ABB RobotStudio station: sesion1.rsstn

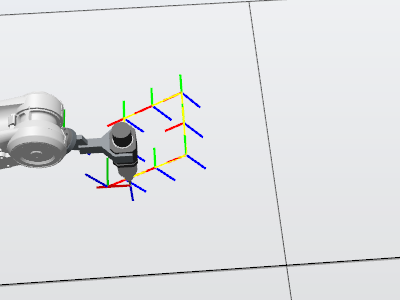
Station sesion1 (saved by RobotStudio 24.1.10713.1)
Controller Controlador1
  mechanical unit ROB_1: IRB140_6_81_C_03, 6 joints, base frame (0, 0, 0) mm
Layout (positions relative to the parent item):
  - IRB140_6_81_C_03 [mechanism, from %ABB.RobotStudio.Models.IRB140%\IRB140_6_81_C_G_03.rslib] at (0, 0, 0) mm; joint values [0, 0.0003, -0.1849, 0, 1.0922, 0] (rad or m)
  - MyTool [mechanism, from Training Objects\myTool.rslib] at (483.67, 0, 730.53) mm, rotated rx 180 ry 38 rz 180 deg
Attachment: MyTool is attached to IRB140_6_81_C_03 / Link6
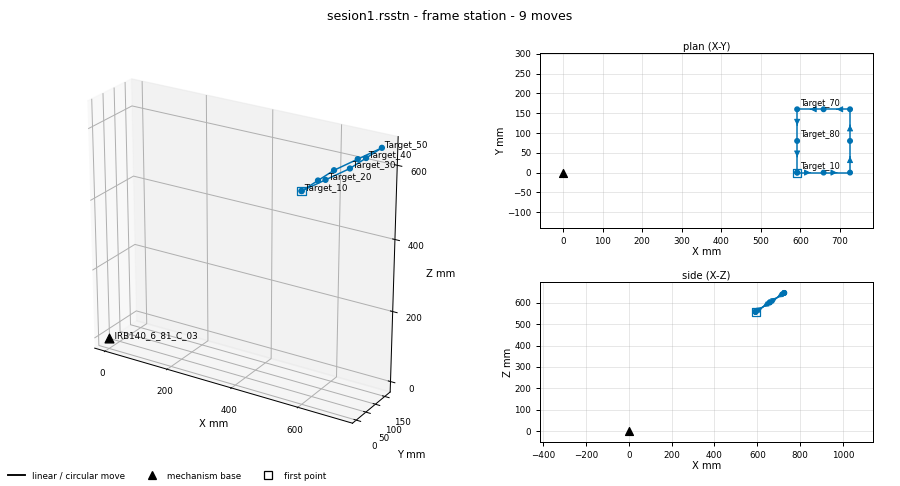
[picture p0: tool path of sesion1.rsstn in frame station, 9 of 9 moves have a stored position in this frame; points joined in program order, loops and branches not executed]
Targets, tools, work objects and paths stored in the station, written as RAPID:
! task T_ROB1
MODULE CalibData
  PERS tooldata MyTool:=[TRUE,[[31.792631019,0,229.638935148],[0.945518576,0,0.325568154,0]],[1,[0,0,1],[1,0,0,0],0,0,0]];
  TASK PERS wobjdata Workobject_1:=[FALSE,TRUE,"",[[550,0,530],[0.957921558,0,-0.287030119,0]],[[0,0,0],[1,0,0,0]]];
ENDMODULE

! task T_ROB1
MODULE Module1
  CONST robtarget Target_10:=[[50,0,0],[0,0,1,0],[0,-1,0,0],[9E+09,9E+09,9E+09,9E+09,9E+09,9E+09]];
  CONST robtarget Target_20:=[[130,0,0],[0,0,1,0],[0,0,-1,0],[9E+09,9E+09,9E+09,9E+09,9E+09,9E+09]];
  CONST robtarget Target_30:=[[210,0,0],[0,0,1,0],[-1,0,-1,0],[9E+09,9E+09,9E+09,9E+09,9E+09,9E+09]];
  CONST robtarget Target_40:=[[210,80,0],[0,0,1,0],[0,-1,0,0],[9E+09,9E+09,9E+09,9E+09,9E+09,9E+09]];
  CONST robtarget Target_50:=[[210,160,0],[0,0,1,0],[0,-1,0,0],[9E+09,9E+09,9E+09,9E+09,9E+09,9E+09]];
  CONST robtarget Target_60:=[[130,160,0],[0,0,1,0],[0,-1,0,0],[9E+09,9E+09,9E+09,9E+09,9E+09,9E+09]];
  CONST robtarget Target_70:=[[50,160,0],[0,0,1,0],[0,-1,0,0],[9E+09,9E+09,9E+09,9E+09,9E+09,9E+09]];
  CONST robtarget Target_80:=[[50,80,0],[0,0,1,0],[0,-1,0,0],[9E+09,9E+09,9E+09,9E+09,9E+09,9E+09]];
  PROC Path_10()
    MoveL Target_10,v50,fine,MyTool\WObj:=Workobject_1;
    MoveL Target_20,v50,fine,MyTool\WObj:=Workobject_1;
    MoveL Target_30,v50,fine,MyTool\WObj:=Workobject_1;
    MoveL Target_40,v50,fine,MyTool\WObj:=Workobject_1;
    MoveL Target_50,v50,fine,MyTool\WObj:=Workobject_1;
    MoveL Target_60,v50,fine,MyTool\WObj:=Workobject_1;
    MoveL Target_70,v50,fine,MyTool\WObj:=Workobject_1;
    MoveL Target_80,v50,fine,MyTool\WObj:=Workobject_1;
    MoveL Target_10,v50,fine,MyTool\WObj:=Workobject_1;
  ENDPROC
ENDMODULE

